INTERFACE I_RecipeBuilder

METHOD Build : BOOL
END_METHOD

PROPERTY Config : ST_RecipeBuilder_Config
GET
END_GET
SET
END_SET
END_PROPERTY

PROPERTY SegmentsCutX : ARRAY [1..32] OF ST_CutSegment
GET
END_GET
END_PROPERTY

PROPERTY SegmentsCutY : ARRAY [1..32] OF ST_CutSegment
GET
END_GET
END_PROPERTY

PROPERTY SegmentsGroove : ARRAY [1..32] OF ST_CutSegment
GET
END_GET
END_PROPERTY

PROPERTY SegmentsToCutX : INT
GET
END_GET
END_PROPERTY

PROPERTY SegmentsToCutY : INT
GET
END_GET
END_PROPERTY

PROPERTY SegmentsToGroove : INT
GET
END_GET
END_PROPERTY

END_INTERFACE

(* stored: Version 1.1.0.1, ProductVersion 3.1.4024.15
   Itf I_RecipeBuilder: Id {a1b2c3d4-1111-4222-b333-c4d5e6f7a8b9}
   Method Build: Id {b2c3d4e5-2222-4333-c444-d5e6f7a8b9c0}
   Property Config: Id {41a1f94d-1ba6-473a-8fd2-d71e6a5c7ac8}
   Get Get: Id {9b92c909-482e-45d4-839d-e73654fca949}
   Set Set: Id {e3c0a41f-b8d2-4dbf-bb3c-74c7ca0bddef}
   Property SegmentsCutX: Id {a7b8c9d0-7777-4888-b999-c0d1e2f3a4b5}
   Get Get: Id {b8c9d0e1-8888-4999-c000-d1e2f3a4b5c6}
   Property SegmentsCutY: Id {e1f2a3b4-bbbb-4ccc-f333-a4b5c6d7e8f9}
   Get Get: Id {f2a3b4c5-cccc-4ddd-a444-b5c6d7e8f9a0}
   Property SegmentsGroove: Id {c3d4e5f6-3333-4444-d555-e6f7a8b9c0d1}
   Get Get: Id {d4e5f6a7-4444-4555-e666-f7a8b9c0d1e2}
   Property SegmentsToCutX: Id {c9d0e1f2-9999-4aaa-d111-e2f3a4b5c6d7}
   Get Get: Id {d0e1f2a3-aaaa-4bbb-e222-f3a4b5c6d7e8}
   Property SegmentsToCutY: Id {a3b4c5d6-dddd-4eee-b555-c6d7e8f9a0b1}
   Get Get: Id {b4c5d6e7-eeee-4fff-c666-d7e8f9a0b1c2}
   Property SegmentsToGroove: Id {e5f6a7b8-5555-4666-f777-a8b9c0d1e2f3}
   Get Get: Id {f6a7b8c9-6666-4777-a888-b9c0d1e2f3a4} *)
